PROGRAM OP90_JB_IO

VAR
	OP90_JB_DI_MODULE_1 AT %I* : WORD;
	OP90_JB_DI_MODULE_2 AT %I* : WORD;
	OP90_JB_DI_MODULE_3 AT %I* : WORD;
	
	OP90_JB_DO_MODULE_1  AT %Q* : WORD;
	OP90_JB_DO_MODULE_2 AT %Q* : WORD;
	
	WORD_AS_BIT_0: WORD_AS_BIT;
	WORD_AS_BIT_1: WORD_AS_BIT;
	WORD_AS_BIT_2: WORD_AS_BIT;
	
	BIT_AS_WORD_0: BIT_AS_WORD;
	BIT_AS_WORD_1: BIT_AS_WORD;
END_VAR

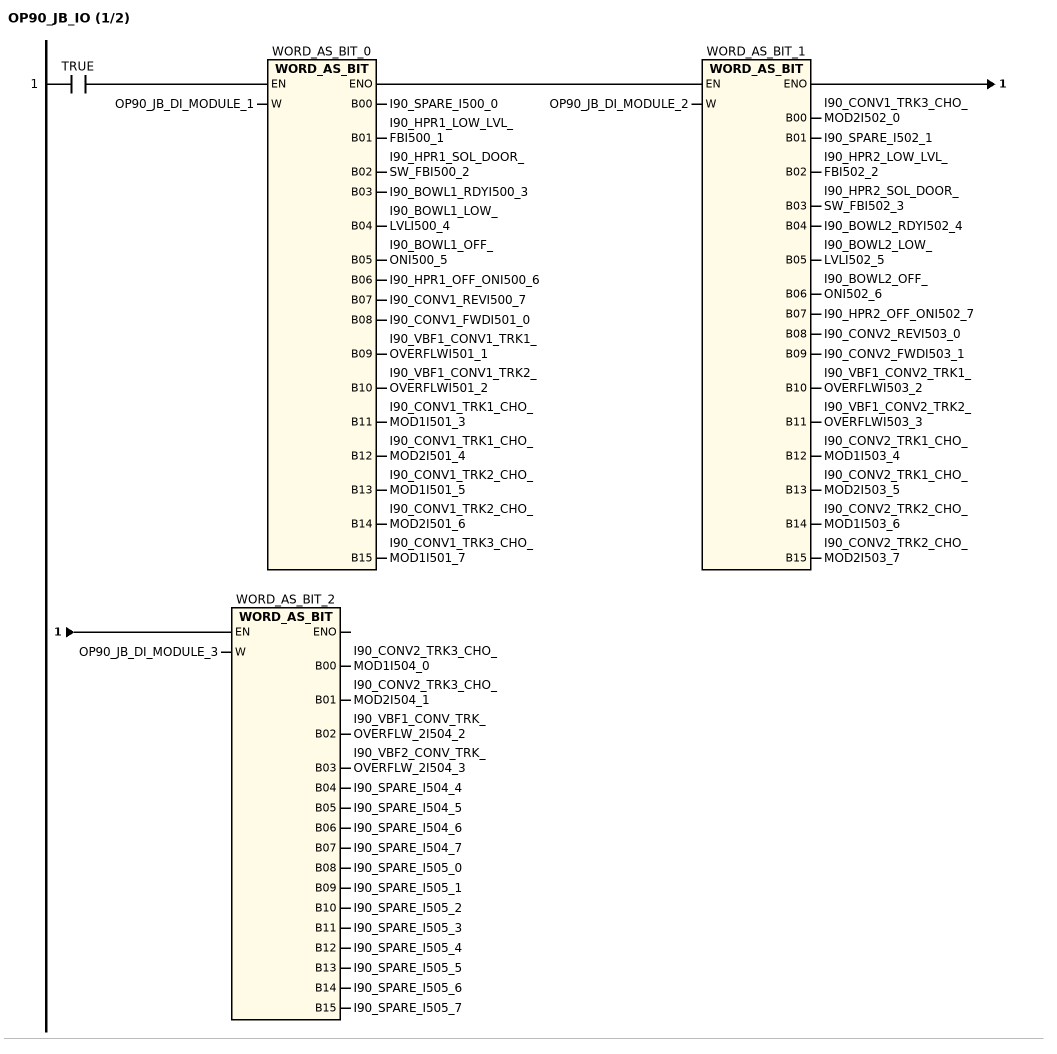
// NETWORK 1
WORD_AS_BIT_0(
    W := OP90_JB_DI_MODULE_1,
    B00 => I90_SPARE_I500_0,
    B01 => I90_HPR1_LOW_LVL_FBI500_1,
    B02 => I90_HPR1_SOL_DOOR_SW_FBI500_2,
    B03 => I90_BOWL1_RDYI500_3,
    B04 => I90_BOWL1_LOW_LVLI500_4,
    B05 => I90_BOWL1_OFF_ONI500_5,
    B06 => I90_HPR1_OFF_ONI500_6,
    B07 => I90_CONV1_REVI500_7,
    B08 => I90_CONV1_FWDI501_0,
    B09 => I90_VBF1_CONV1_TRK1_OVERFLWI501_1,
    B10 => I90_VBF1_CONV1_TRK2_OVERFLWI501_2,
    B11 => I90_CONV1_TRK1_CHO_MOD1I501_3,
    B12 => I90_CONV1_TRK1_CHO_MOD2I501_4,
    B13 => I90_CONV1_TRK2_CHO_MOD1I501_5,
    B14 => I90_CONV1_TRK2_CHO_MOD2I501_6,
    B15 => I90_CONV1_TRK3_CHO_MOD1I501_7); // WORD_AS_BIT
WORD_AS_BIT_1(
    W := OP90_JB_DI_MODULE_2,
    B00 => I90_CONV1_TRK3_CHO_MOD2I502_0,
    B01 => I90_SPARE_I502_1,
    B02 => I90_HPR2_LOW_LVL_FBI502_2,
    B03 => I90_HPR2_SOL_DOOR_SW_FBI502_3,
    B04 => I90_BOWL2_RDYI502_4,
    B05 => I90_BOWL2_LOW_LVLI502_5,
    B06 => I90_BOWL2_OFF_ONI502_6,
    B07 => I90_HPR2_OFF_ONI502_7,
    B08 => I90_CONV2_REVI503_0,
    B09 => I90_CONV2_FWDI503_1,
    B10 => I90_VBF1_CONV2_TRK1_OVERFLWI503_2,
    B11 => I90_VBF1_CONV2_TRK2_OVERFLWI503_3,
    B12 => I90_CONV2_TRK1_CHO_MOD1I503_4,
    B13 => I90_CONV2_TRK1_CHO_MOD2I503_5,
    B14 => I90_CONV2_TRK2_CHO_MOD1I503_6,
    B15 => I90_CONV2_TRK2_CHO_MOD2I503_7); // WORD_AS_BIT
WORD_AS_BIT_2(
    W := OP90_JB_DI_MODULE_3,
    B00 => I90_CONV2_TRK3_CHO_MOD1I504_0,
    B01 => I90_CONV2_TRK3_CHO_MOD2I504_1,
    B02 => I90_VBF1_CONV_TRK_OVERFLW_2I504_2,
    B03 => I90_VBF2_CONV_TRK_OVERFLW_2I504_3,
    B04 => I90_SPARE_I504_4,
    B05 => I90_SPARE_I504_5,
    B06 => I90_SPARE_I504_6,
    B07 => I90_SPARE_I504_7,
    B08 => I90_SPARE_I505_0,
    B09 => I90_SPARE_I505_1,
    B10 => I90_SPARE_I505_2,
    B11 => I90_SPARE_I505_3,
    B12 => I90_SPARE_I505_4,
    B13 => I90_SPARE_I505_5,
    B14 => I90_SPARE_I505_6,
    B15 => I90_SPARE_I505_7); // WORD_AS_BIT

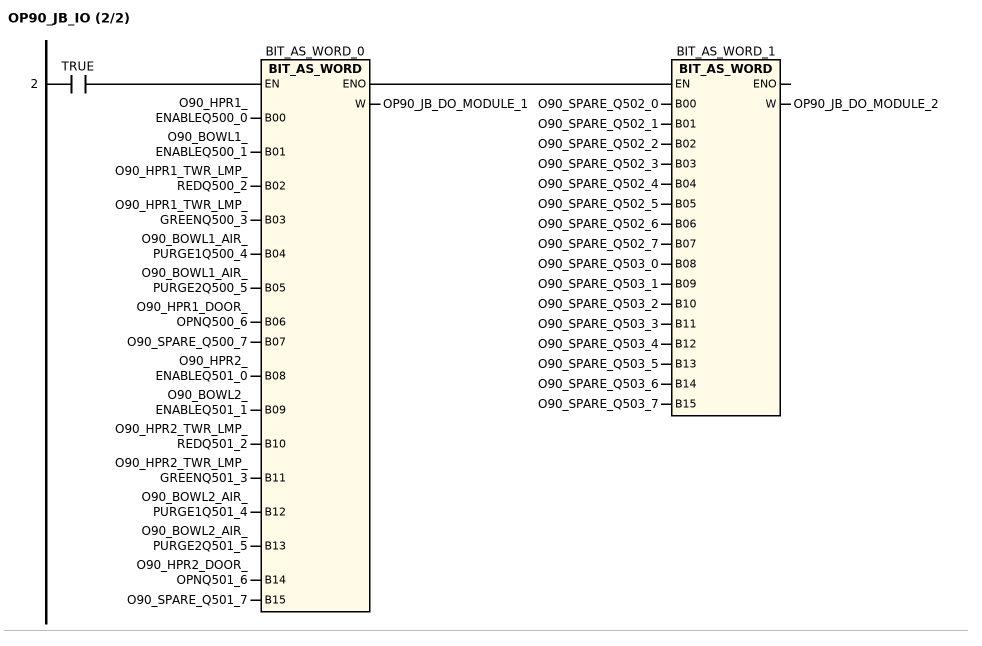
// NETWORK 2
BIT_AS_WORD_0(
    B00 := O90_HPR1_ENABLEQ500_0,
    B01 := O90_BOWL1_ENABLEQ500_1,
    B02 := O90_HPR1_TWR_LMP_REDQ500_2,
    B03 := O90_HPR1_TWR_LMP_GREENQ500_3,
    B04 := O90_BOWL1_AIR_PURGE1Q500_4,
    B05 := O90_BOWL1_AIR_PURGE2Q500_5,
    B06 := O90_HPR1_DOOR_OPNQ500_6,
    B07 := O90_SPARE_Q500_7,
    B08 := O90_HPR2_ENABLEQ501_0,
    B09 := O90_BOWL2_ENABLEQ501_1,
    B10 := O90_HPR2_TWR_LMP_REDQ501_2,
    B11 := O90_HPR2_TWR_LMP_GREENQ501_3,
    B12 := O90_BOWL2_AIR_PURGE1Q501_4,
    B13 := O90_BOWL2_AIR_PURGE2Q501_5,
    B14 := O90_HPR2_DOOR_OPNQ501_6,
    B15 := O90_SPARE_Q501_7,
    W => OP90_JB_DO_MODULE_1); // BIT_AS_WORD
BIT_AS_WORD_1(
    B00 := O90_SPARE_Q502_0,
    B01 := O90_SPARE_Q502_1,
    B02 := O90_SPARE_Q502_2,
    B03 := O90_SPARE_Q502_3,
    B04 := O90_SPARE_Q502_4,
    B05 := O90_SPARE_Q502_5,
    B06 := O90_SPARE_Q502_6,
    B07 := O90_SPARE_Q502_7,
    B08 := O90_SPARE_Q503_0,
    B09 := O90_SPARE_Q503_1,
    B10 := O90_SPARE_Q503_2,
    B11 := O90_SPARE_Q503_3,
    B12 := O90_SPARE_Q503_4,
    B13 := O90_SPARE_Q503_5,
    B14 := O90_SPARE_Q503_6,
    B15 := O90_SPARE_Q503_7,
    W => OP90_JB_DO_MODULE_2); // BIT_AS_WORD

END_PROGRAM

(* stored: Version 1.1.0.1, ProductVersion 3.1.4024.11
   POU OP90_JB_IO: Id {d4edafc1-797d-4162-878c-8314fe11a878}, SpecialFunc None *)
